FUNCTION_BLOCK TestTransition
  (* Standard: 61499-2 *)
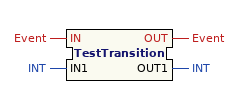
  EVENT_INPUT
    IN;
  END_EVENT
  EVENT_OUTPUT
    OUT;
  END_EVENT
  VAR_INPUT
    IN1 : INT;
  END_VAR
  VAR_OUTPUT
    OUT1 : INT;
  END_VAR
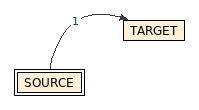
  EC_STATES
    SOURCE;
    TARGET;
  END_STATES
  EC_TRANSITIONS
    SOURCE TO TARGET := 1;
  END_TRANSITIONS
END_FUNCTION_BLOCK
